(*
Info!
*)
FUNCTION_BLOCK FB_MyBlock
VAR_INPUT
    someInput       : LREAL;        // This is some input with a description
    otherInput      : BOOL;         // Awesome description 
END_VAR
VAR_INPUT
    secondClause    : LREAL;        // This is some input with a description 
END_VAR
VAR_OUTPUT
    myOutput        : UINT;         // Return something nice
END_VAR
VAR
END_VAR

myOutput := 420;

METHOD AnotherMethod : LREAL
VAR_INPUT
    methodInput     : LREAL;            // Some input
END_VAR
END_METHOD

(*
This is a description.
*)
METHOD MyMethod : BOOL
VAR_INPUT
END_VAR
MyMethod := FALSE;
END_METHOD

END_FUNCTION_BLOCK

(* stored: Version 1.1.0.1, ProductVersion 3.1.4024.11
   POU FB_MyBlock: Id {349377b9-c8f5-4136-9f25-4b51249737ae}, SpecialFunc None
   Method AnotherMethod: Id {1f1a001e-6f51-4979-b89d-4d72f4734951}
   Method MyMethod: Id {0c39134c-0d9c-4e67-a24c-81526057b12e} *)
